FUNCTION_BLOCK Servo
VAR
	mqttSettings : MQTTSettings;	

	currentSpeed : INT;
	currentAngle : INT;
	
	servoAngleCommandTopic : STRING := 'plc/servo/angle';
	servoAngleOutTopic : STRING := 'plc/servo/angle/out';
	servoSpeedOutTopic : STRING := 'plc/servo/speed/out';
	isSubscribed : BOOL := FALSE;
END_VAR

METHOD getAngle : INT
VAR_OUTPUT
	angle : INT;
END_VAR
angle := currentAngle;
END_METHOD

METHOD publishAngle
VAR_IN_OUT
	mqtt: MQTT;	
	timer : TON;
END_VAR
IF mqtt.isConnected() THEN
    timer(IN:=TRUE);
    IF timer.Q THEN
        timer(IN:=FALSE);
        mqtt.publishToTopic(topic := servoAngleOutTopic, msg := INT_TO_STRING(currentAngle));
    END_IF
END_IF
END_METHOD

METHOD publishSpeed
VAR_IN_OUT
	mqtt: MQTT;	
	timer : TON;
END_VAR
IF mqtt.isConnected() THEN
    timer(IN:=TRUE);
    IF timer.Q THEN
        timer(IN:=FALSE);
        mqtt.publishToTopic(topic := servoSpeedOutTopic, msg := INT_TO_STRING(currentSpeed));
    END_IF
END_IF
END_METHOD

METHOD setAngle : BOOL
VAR_INPUT
	angleToSet : INT;
END_VAR
currentAngle := angleToSet;
END_METHOD

METHOD waitForCommand
VAR_IN_OUT
	mqtt: MQTT;	
END_VAR
VAR
	receivedMsg : STRING(255);
	
	angleToSet : INT;
END_VAR
IF mqtt.isConnected() THEN
	IF NOT isSubscribed THEN
        isSubscribed := mqtt.mqttClient.Subscribe(sTopic:=servoAngleCommandTopic, eQoS:=mqttSettings.qos);
    END_IF	

	IF mqtt.messageQueue.nQueuedMessages > 0 THEN	
		IF mqtt.messageQueue.Dequeue(fbMessage:=mqtt.message) THEN
			IF mqtt.message.CompareTopic(sTopic:=servoAngleCommandTopic) THEN	
	
				mqtt.message.GetPayload(pPayload:=ADR(receivedMsg), nPayloadSize:=SIZEOF(receivedMsg), bSetNullTermination:=FALSE);				
				angleToSet := STRING_TO_INT(receivedMsg);
				IF (angleToSet >= 0 AND angleToSet <= 360) THEN
					setAngle(angleToSet := angleToSet);
				END_IF
			
			END_IF
		END_IF
	END_IF
	
END_IF
END_METHOD

END_FUNCTION_BLOCK

(* stored: Version 1.1.0.1, ProductVersion 3.1.4024.12
   POU Servo: Id {8e476ada-403f-4aab-b2d0-f33c8df5abc6}, SpecialFunc None
   Method getAngle: Id {fcf94f04-c45b-4525-965b-43b1879cd6c3}
   Method publishAngle: Id {90aeb0ea-dcee-414a-9650-a99ab35755f5}
   Method publishSpeed: Id {ad9a4890-ffc5-45db-960e-ecf23fd083a0}
   Method setAngle: Id {efa850a3-5964-414f-b9ff-7d6606d6fd36}
   Method waitForCommand: Id {a3edf7ce-7614-4fe1-bb56-cf52d65bc955} *)
